{attribute 'qualified_only'}
// Simulated I/O Outputs
//
VAR_GLOBAL

	// Simulated output signals...
	o_HtrTemp AT %Q*: REAL; // Heater temperature [°C]
 
END_VAR

(* stored: Version 1.1.0.1, ProductVersion 3.1.4022.6
   GVL IO_Outputs: Id {f0a1e0a0-6166-4e5c-80ff-9aa7e9099178} *)
